(* CoDeSys 2.3.9.41 project: testmodbus.pro *)
(* Libraries: Util.lib 18.5.10 15:14:28, ПЛК_ПЧВ_v2.lib 26.7.19 14:18:06, STANDARD.LIB 4.10.05 11:14:46, IECSFC.LIB 13.4.06 15:51:28, ANALYZATION.LIB 5.10.99 09:05:06 *)

(* PLC configuration (modules and I/O channels)
InputByte AT %IB0.0 [ByteInput] 8 discrete inputs
Discrete output 2 bit [ID101] node 1, in %IB1 out %QB1 {PinCount = 2; SafeValueBool = FALSE; SafeValueBool = FALSE; Visibility = No}
  DO_1_0 AT %QX1.0 [BitOutput] First
  DO_1_1 AT %QX1.1 [BitOutput] Second
Discrete output 2 bit [ID101] node 2, in %IB2 out %QB2 {PinCount = 2; SafeValueBool = FALSE; SafeValueBool = FALSE; Visibility = No}
  DO_2_0 AT %QX2.0 [BitOutput] First
  AT %QX2.1 [BitOutput] Second
Discrete output 2 bit [ID101] node 3, in %IB3 out %QB3 {PinCount = 2; SafeValueBool = FALSE; SafeValueBool = FALSE; Visibility = No}
  DO_3_0 AT %QX3.0 [BitOutput] First
  AT %QX3.1 [BitOutput] Second
Discrete output 2 bit [ID101] node 4, in %IB4 out %QB4 {PinCount = 2; SafeValueBool = FALSE; SafeValueBool = FALSE; Visibility = No}
  DO_4_0 AT %QX4.0 [BitOutput] First
  AT %QX4.1 [BitOutput] Second
Discrete output 2 bit [ID101] node 5, in %IB5 out %QB5 {PinCount = 2; SafeValueBool = FALSE; SafeValueBool = FALSE; Visibility = No}
  DO_5_0 AT %QX5.0 [BitOutput] First
  AT %QX5.1 [BitOutput] Second
Discrete output 2 bit [ID101] node 6, in %IB6 out %QB6 {PinCount = 2; SafeValueBool = FALSE; SafeValueBool = FALSE; Visibility = No}
  DO_6_0 AT %QX6.0 [BitOutput] First
  AT %QX6.1 [BitOutput] Second
Special output [ID104] node 7, in %IB7 out %QB7 {Visibility = No; PinCount = 1}
  AT %QX7.0 [BitOutput] Special output
ModBus (Master) [MODBUS_MASTER_ID450] node 8, in %IB8 out %QB8 {Visibility = No}
  modbusLastAddr AT %QD8.0 [DWordOutput] Last address
  modbusLastErr AT %QW8.1 [WordOutput] Last error
  RS-485-1 [COM1_USART] node 0, in %IB8.0 out %QB8.0 {CommunicationSpeed = 19200; Parity = NO PARITY CHECK; BitLength = 8 bits; StopLength = One stop bit; InterfaceType = RS485; FrameOriented = RTU; Timeout = 0; Visibility = No}
  Universal Modbus device [ID2000] node 1, in %IB8.1 out %QB8.1 {ModuleIP = 10:0:0:223; ServiceTimeout = 150; TCPport = 502; NetMode = Serial; ModuleSlaveAddress = 2; RequestType = By poll time; PeriodOfService = 1000; Visibility = No; RepeatCounter = 2; ByteSequence = Native}
    AT %QB8.1.0 [ComChannel] Command (0xff - Start)
Dist_on_pistol_1 AT %IW8.1.0.0 [WordInput]
Dist_on_pistol_2 AT %IW8.1.1.0 [WordInput]
Dist_on_pistol_3 AT %IW8.1.2.0 [WordInput]
Dist_on_pistol_4 AT %IW8.1.3.0 [WordInput]
Dist_on_pistol_5 AT %IW8.1.4.0 [WordInput]
Dist_on_pistol_6 AT %IW8.1.5.0 [WordInput]
Dist_on_pistol_7 AT %IW8.1.6.0 [WordInput]
Dist_on_pistol_8 AT %IW8.1.7.0 [WordInput]
Dist_off_pistol_1 AT %IW8.1.8.0 [WordInput]
Dist_off_pistol_2 AT %IW8.1.9.0 [WordInput]
Dist_off_pistol_3 AT %IW8.1.10.0 [WordInput]
Dist_off_pistol_4 AT %IW8.1.11.0 [WordInput]
Dist_off_pistol_5 AT %IW8.1.12.0 [WordInput]
Dist_off_pistol_6 AT %IW8.1.13.0 [WordInput]
Dist_off_pistol_7 AT %IW8.1.14.0 [WordInput]
Dist_off_pistol_8 AT %IW8.1.15.0 [WordInput]
DistOnPistMinimum AT %IW8.1.16.0 [WordInput]
qInvStatusW AT %QW8.1.17.0 [WordOutput]
Universal Modbus device [ID2000] node 2, in %IB8.2 out %QB8.2 {ModuleIP = 10:0:0:223; ServiceTimeout = 150; TCPport = 502; NetMode = Serial; ModuleSlaveAddress = 2; RequestType = By poll time; PeriodOfService = 1500; Visibility = No; RepeatCounter = 2; ByteSequence = Native}
  AT %QB8.2.0 [ComChannel] Command (0xff - Start)
iTP1 AT %IW8.2.0.0 [WordInput]
iTP2 AT %IW8.2.1.0 [WordInput]
iTP3 AT %IW8.2.2.0 [WordInput]
iTP4 AT %IW8.2.3.0 [WordInput]
iTP5 AT %IW8.2.4.0 [WordInput]
iTP6 AT %IW8.2.5.0 [WordInput]
iTP7 AT %IW8.2.6.0 [WordInput]
iTP8 AT %IW8.2.7.0 [WordInput]
iTPGlob AT %ID8.2.8.0 [FloatInput]
Universal Modbus device [ID2000] node 3, in %IB8.3 out %QB8.3 {ModuleIP = 10:0:0:223; ServiceTimeout = 150; TCPport = 502; NetMode = Serial; ModuleSlaveAddress = 2; RequestType = By poll time; PeriodOfService = 700; Visibility = No; RepeatCounter = 2; ByteSequence = Native}
  AT %QB8.3.0 [ComChannel] Command (0xff - Start)
task_speed_panel_real AT %ID8.3.0.0 [FloatInput]
speed_at_50Hz AT %ID8.3.1.0 [FloatInput]
speed_at_25Hz AT %ID8.3.2.0 [FloatInput]
speed_Max_panel AT %ID8.3.3.0 [FloatInput]
speed_Min_panel AT %ID8.3.4.0 [FloatInput]
qDetR AT %ID8.3.5.0 [FloatInput]
qMetR AT %ID8.3.6.0 [FloatInput]
follow_Sign_Loss AT %IW8.3.7.0 [WordInput]
qMaxDetLen AT %IW8.3.8.0 [WordInput]
qVersion AT %QD8.3.9.0 [FloatOutput]
Universal Modbus device [ID2000] node 4, in %IB8.4 out %QB8.4 {ModuleIP = 10:0:0:223; ServiceTimeout = 150; TCPport = 502; NetMode = Serial; ModuleSlaveAddress = 2; RequestType = By value change; PeriodOfService = 100; Visibility = No; RepeatCounter = 2; ByteSequence = Native}
  AT %QB8.4.0 [ComChannel] Command (0xff - Start)
qInputB_DO1_6 AT %QW8.4.0.0 [WordOutput]
Universal Modbus device [ID2000] node 5, in %IB8.5 out %QB8.5 {ModuleIP = 10:0:0:223; ServiceTimeout = 150; TCPport = 502; NetMode = Serial; ModuleSlaveAddress = 2; RequestType = By poll time; PeriodOfService = 200; Visibility = No; RepeatCounter = 2; ByteSequence = Native}
  AT %QB8.5.0 [ComChannel] Command (0xff - Start)
qStatusW AT %QW8.5.0.0 [WordOutput]
controlPing AT %ID8.5.1.0 [FloatInput]
qDet_met AT %QD8.5.2.0 [FloatOutput]
qDet_Cnt AT %QD8.5.3.0 [FloatOutput]
controlPong AT %QD8.5.4.0 [FloatOutput]
qAbuseW AT %IW8.5.5.0 [WordInput]
qlast_Det_Len AT %QD8.5.6.0 [FloatOutput]
qlast_Det_Time AT %QD8.5.7.0 [FloatOutput]
AT %QB8.6.0 [ComChannel] Command (0xff - Start)
Status_word AT %IW8.6.0.0 [WordInput]
Frequency AT %IW8.6.1.0 [WordInput]
Power AT %IW8.6.2.0 [WordInput]
Voltage AT %IW8.6.3.0 [WordInput]
Current AT %IW8.6.4.0 [WordInput]
Inv_Error AT %ID8.6.5.0 [DWordInput]
Minimum_frequency AT %IW8.6.6.0 [WordInput]
Maximum_frequency AT %IW8.6.7.0 [WordInput]
Command_word AT %QW8.6.8.0 [WordOutput]
Task_RS485 AT %IW8.6.9.0 [WordInput]
Set_Speed AT %QW8.6.10.0 [WordOutput] 0-16384
Set_MinTask AT %QD8.6.11.0 [DWordOutput]
Set_MaxTask AT %QD8.6.12.0 [DWordOutput]
*)

(* Task configuration *)
TASK cycle_counters (PRIORITY := 0, INTERVAL := T#5ms);
	counters();
END_TASK
TASK main_task (PRIORITY := 1); (* freewheeling *)
	PLC_PRG();
END_TASK

(* Global variable list: Global_Variables *)
VAR_GLOBAL
	total_cycles: DWORD;
	details_meters: REAL;			(*прошло деталей в метрах - берётся от длины в мм*)
	contr_StatusW:  WORD;   			(*статусное слово контроллера - заполняем в главном цикле*)
	contr_AbuseW: WORD;			(*командное слово контроллера - отрабатывает в главном цикле*)
       needSynhro : BOOL := TRUE;	(*Если требуется синхронизация - конвейер не обрабатывает команды управления*)
	freeCounters: BOOL := TRUE;	(*приказ очистить массив счетчика и ВЫКЛючить Пистолеты*)
	last_Limit_switch_part: BOOL := FALSE; (*предыдущее значение датчика детали*)
	last_Det_length: REAL := 0.0;
	last_Det_Time: REAL := 0.0;		(*последнее время на деталь в миллисекундах*)
	version: REAL := 0.6;
	pist: ARRAY[1..4] OF BOOL;
END_VAR

VAR_GLOBAL   (*переменные ошибок*)
	errSensor: BOOL := FALSE; 		(* вырабатывается если количество деталей превысило Максимум или слишком длинная деталь *)
										(* пока активна ошибка - не будут накапливаться данные о деталях, пистолеты выключатся*)
	errTaskSpeed: BOOL := FALSE; 	(* вырабатывается если значение скорости не в диапазоне макс/мин или равно 0 *)

END_VAR

VAR_GLOBAL
	(*Входы контроллера*)
	Start_conveyor: BOOL;    			(*DI_1 Включить конвейер *)
	Stop_conveyor: BOOL;   			(*DI_2 Выключить конвейер *)
	Following_machine: BOOL;   		(*DI_3 Сигнал от следующей машины*)
	Fan_on: BOOL;					(*DI_4 Вытяжка включена*)
	(*Pistols_automat_mode: BOOL;	Пистолеты в автоматическом режиме*)
	Door_Closed: BOOL;				(*DI_5 Концевой выключатель двери*)
	Limit_switch_part: BOOL;			(*DI_6 Концевой выключатель наличия детали*)
	Pistols_5_8_run: BOOL;			(*DI_7 Включены пистолеты 5-8*)

	(*Выходы контроллера*)
	Conveyor_green: BOOL;                     (*Конвейер готов к включению (сигнальная лампа) *)
	Conveyor_runNow: BOOL;			(*Конвейер поехал,сигнал на предыдущую машину *)

END_VAR

VAR_GLOBAL RETAIN PERSISTENT (*эти данные хранятся в энергонезависимой памяти*)
	details_count: REAL;				(*Счётчик кол-ва деталей. Сбрасывается по команде с панели *)
	details_mMeters: REAL;			(*Счётчик общей длины детали в мм, сбрасывается с панели *)
	details_Real_mMeters: REAL;	(*Необнуляемый счётчик  общей длины детали в мм*)
END_VAR

(* POU counters, ST *)
PROGRAM counters
VAR CONSTANT
	MAXDETCNT:INT:= 10;
END_VAR

VAR
	cycleinterval_ms: REAL := 4.99; (*такой установлен в конфигураторе задач !!!!!!!!!!!!!!!!!!!!!!!!!!!!!!!!!!!!!!!!!!!!!!!!!!!!!!!!!!!!!!!!!!!!*)

   (*    cycleinterval_ms_calc: REAL;
	lasttime: TIME;
	total_cycles_loss: DWORD; *)

	cycle_mm: REAL; (*надо пересчитать в мм на текущий момент времени в зависимости от скорости погонажки*)
	Counter: ARRAY[1..4, 0..1, 0..MAXDETCNT] OF REAL; (* 4 pistools, On(0), Off(1), push counter     in mm ! *)
	PistLen: ARRAY[1..4,0..1] OF INT; (*4 pist, 0 - Up Len, 1 - UpLen+Off Len *)
	PistTime: ARRAY[1..4] OF INT; (*время предварительного срабатывания пистолета - пересчёт в мм*)
	i,j,k: INT;
	detOn: BOOL;
	detOff: BOOL;
	need_Pistols_On: BOOL;
END_VAR
(*программа выполняется с частотой вызовов 1 раз в 5 мсек*)
(*m/min > *)
(*cycleinterval_ms_calc := TIME_TO_REAL(TIME()-lastTime)+0.01;
lastTime := TIME();*)
(*
CycleTime_100mks;
CPU_OverLoaded;

total_cycles := total_cycles+1;
total_cycles_loss := total_cycles_loss + BOOL_TO_DWORD( cycleinterval_ms <> cycleInterval_ms_calc);
*)
cycle_mm := task_speed_panel_real*1000/60/(1000/cycleinterval_ms);

	FOR i := 1 TO 4 DO
	FOR j := 0 TO 1 DO
		FOR k:=0 TO MAXDETCNT DO
			IF freecounters THEN
				Counter[i,j,k] := 0.0;
			END_IF;
		END_FOR
	END_FOR
	IF freecounters THEN
		Counter[i,1,0] := 0.001; (*выключить пистолет*)
	END_IF;
	END_FOR
	freecounters := FALSE;

Limit_switch_part:=DI_6 AND NOT errSensor; 	(*Концевой выключатель наличия детали причём если нет его ошибки*)
Pistols_5_8_run:=DI_7; 	(*Включены пистолеты 5-8*)

(*прошел цикл, значит пора сократить все длины на cycle_mm, заодно разобраться с включением выключением,
а потом уже сделать перенос величин ставших менее 0.0*)

FOR i := 1 TO 4 DO
	FOR j := 0 TO 1 DO
		FOR k:=0 TO MAXDETCNT DO
			IF Counter[i,j,k] <> 0.0 THEN
				Counter[i,j,k] := Counter[i,j,k]-cycle_mm;
			END_IF;
		END_FOR
	END_FOR
								  (* СПЕРВА ВЫКЛЮЧИМ, ПОТОМ ВКЛЮЧИМ - убираем пересечения *)
	IF (Counter[i,1,0] < 0)  THEN (*начало  цикла (голова) в нуле. если нулевое стало меньше 1 - выключим пистолет, но не если есть след.деталь*)
		pist[i] := FALSE;
	END_IF;
	IF Counter[i,0,0] < 0 THEN (*начало  цикла (голова) в нуле. если нулевое стало меньше 0 - включим пистолет*)
		pist[i] := TRUE;
	END_IF;
END_FOR

detOn := FALSE;
detOff := FALSE;

IF NOT last_Limit_switch_part AND Limit_switch_part THEN (*деталь началась*)
	detOn := TRUE;
	last_Det_length := 0.0;
	last_Det_time := 0.0;
END_IF;

IF last_Limit_switch_part AND NOT Limit_switch_part THEN (*деталь прошла*)
	details_count := details_count +1;
	qLast_Det_time := last_Det_time;
	detOff := TRUE;
END_IF;

IF Limit_switch_part THEN (*если концевик показывает деталь - увеличим погонаж*)
	details_mMeters := details_mMeters+cycle_mm;
	details_Real_mMeters := details_Real_mMeters +cycle_mm;
	last_Det_Length := last_Det_Length+cycle_mm;
	last_Det_Time := last_Det_Time + cycleinterval_ms;
	IF last_Det_Length > qmaxDetLen THEN
		errSensor := TRUE;
	END_IF;
END_IF;
details_meters := details_mMeters / 1000;

(* заполнить массив включения выключения если не синхронизация *)
IF NOT needSynhro THEN
IF NOT Pistols_5_8_run THEN
   PistLen[1,0] := Dist_on_pistol_1; PistLen[1,1] := Dist_off_pistol_1;
   PistLen[2,0] := Dist_on_pistol_2; PistLen[2,1] := Dist_off_pistol_2;
   PistLen[3,0] := Dist_on_pistol_3; PistLen[3,1] := Dist_off_pistol_3;
   PistLen[4,0] := Dist_on_pistol_4; PistLen[4,1] := Dist_off_pistol_4;
	PistTime[1] := REAL_TO_INT((-INT_TO_REAL(iTP1)+iTPGlob)*cycle_mm/cycleinterval_ms);
	PistTime[2] := REAL_TO_INT((-INT_TO_REAL(iTP2)+iTPGlob)*cycle_mm/cycleinterval_ms);
	PistTime[3] := REAL_TO_INT((-INT_TO_REAL(iTP3)+iTPGlob)*cycle_mm/cycleinterval_ms);
	PistTime[4] := REAL_TO_INT((-INT_TO_REAL(iTP4)+iTPGlob)*cycle_mm/cycleinterval_ms);
ELSE
   PistLen[1,0] := Dist_on_pistol_5; PistLen[1,1] := Dist_off_pistol_5;
   PistLen[2,0] := Dist_on_pistol_6; PistLen[2,1] := Dist_off_pistol_6;
   PistLen[3,0] := Dist_on_pistol_7; PistLen[3,1] := Dist_off_pistol_7;
   PistLen[4,0] := Dist_on_pistol_8; PistLen[4,1] := Dist_off_pistol_8;
	PistTime[1] := REAL_TO_INT((-INT_TO_REAL(iTP5)+iTPGlob)*cycle_mm/cycleinterval_ms);
	PistTime[2] := REAL_TO_INT((-INT_TO_REAL(iTP6)+iTPGlob)*cycle_mm/cycleinterval_ms);
	PistTime[3] := REAL_TO_INT((-INT_TO_REAL(iTP7)+iTPGlob)*cycle_mm/cycleinterval_ms);
	PistTime[4] := REAL_TO_INT((-INT_TO_REAL(iTP8)+iTPGlob)*cycle_mm/cycleinterval_ms);
END_IF;

FOR i := 1 TO 4 DO
IF PistLen[i,0] > 0 THEN (*хоть какая-то длина указана, ок*)
   PistLen [i,0] := PistLen[i,0] + PistTime[i];
   IF PistLen[i,0] <=0 THEN PistLen[i,0] := 1;END_IF;
   PistLen[i,1] := PistLen[i,0] + PistLen[i,1];
END_IF;
END_FOR;

END_IF;

(*прокрутить списки деталей*)

FOR i := 1 TO 4 DO
	j := 0;
	IF Counter[i,j,0] < INT_TO_REAL( PistLen[i,0] - PistLen[i,1])-5.0 THEN (*убрать деталь*)
		FOR k:=0 TO MAXDETCNT-1 DO (*-1, т.к. [,,k] элемент = 0, удобненько*)
			Counter[i,j,k] := Counter[i,j,k+1];
		END_FOR
	END_IF
END_FOR

FOR i := 1 TO 4 DO
	j := 1;
	IF Counter[i,j,0] < 0 THEN (*убрать деталь*)
		FOR k:=0 TO MAXDETCNT-1 DO (*-1, т.к. [,,k] элемент = 0, удобненько*)
			Counter[i,j,k] := Counter[i,j,k+1];
		END_FOR
	END_IF
END_FOR

(*добавить деталь если началась*)
IF detOn THEN
	FOR i := 1 TO 4 DO
	 j := 0;
	FOR k:=0 TO MAXDETCNT-1 DO
		IF Counter[i,j,k] = 0.0 THEN
			EXIT;
		END_IF;
	END_FOR
	(*хочется не добавлять если k - крайний и выработать ошибку*)
	IF k=MAXDETCNT THEN
		errSensor := TRUE;
	ELSE
		Counter[i,j,k] := PistLen[i,0]; (*значение ожидания до включения если оно больше чем DistOnPistMinimum*)
		IF PistLen[i,0] < DistOnPistMinimum THEN  Counter[i,j,k] := 0.0; END_IF;
	END_IF;
	END_FOR
END_IF;

(*добавить конец детали деталь если кончилась*)
IF detOff THEN
	FOR i := 1 TO 4 DO
	 j := 1;
	FOR k:=0 TO MAXDETCNT-1 DO
		IF Counter[i,j,k] = 0.0 THEN
			EXIT;
		END_IF;
	END_FOR
	(*хочется не добавлять если k - крайний и выработать ошибку*)
	IF k=MAXDETCNT THEN
		errSensor := TRUE;
	ELSE
		IF (k > 0) AND (PistLen[i,0] < REAL_TO_INT(Counter[i,j,k-1]) ) THEN (*более 1 детали и перекрывает расстояние, правим предыдущую*)
		   k := k-1;
		END_IF;
		Counter[i,j,k] := PistLen[i,1]; (*значение ожидания до выключения если включение больше чем DistOnPistMinimum*)
		IF PistLen[i,0] < DistOnPistMinimum THEN  Counter[i,j,k] := 0.0; END_IF;
	END_IF;
	END_FOR
END_IF;

need_Pistols_On := contr_abuseW.1  AND Door_Closed AND Fan_on; (*просит включить распыление и ВЫтяжка *)

(*включить/выключить пистолеты *)
DO_3_0 := pist[1] OR need_Pistols_On;
DO_4_0 := pist[2] OR need_Pistols_On;
DO_5_0 := pist[3] OR need_Pistols_On;
DO_6_0 := pist[4] OR need_Pistols_On;

(*запомнить состояние детали*)
last_Limit_switch_part := Limit_switch_part;
END_PROGRAM

(* POU PLC_PRG, ST *)
PROGRAM PLC_PRG
VAR
	synhroW: DWORD := 0;

	com_word: com_word_fb;
	Invertor_stop: BOOL := FALSE;
	Invertor_start: BOOL := FALSE;
	Invertor_reverse:BOOL := FALSE;
	Invertor_speed_ok: BOOL := FALSE;

(*переменные объединяющиес текущий статус контроллера*)
	Invertor_Pwr_On: BOOL := FALSE; (*инвертор найден по шине, получен статус отличный от 0 и он в автомате и готов*)
	Conveyor_On: BOOL; (*включен двигатель конвейера*)

(*просто какие-то временные переменные*)
	w1: WORD;
	dw, mit, mat: DWORD;
	bol: BOOL;
	b: REAL;
	k: REAL;
	modbusInvLastErr: WORD := 0;

(* Статус частотника *)
	stat_word: stat_word_fb;

	Invertor_alarm: BOOL;		(* Авария частотника *)
	Invertor_warning: BOOL; 		(* Предупреждение частотника *)
	Invertor_auto: BOOL;			(* Частотник в автоматическом режиме *)
	Invertor_work: BOOL; 			(* Частотник в работе *)

(*переменные для управления ПЧВ*)
	rsp : REAL;
	abuse_50Hz: BOOL; (*принуждает ПЧВ запустить двигатель на 50 Hz*)
	abuse_25Hz: BOOL; (*принуждает ПЧВ запустить двигатель на 25 Hz*)
	frequency_Equal: BOOL := FALSE;
	lastFreqReqw: WORD := 0;
	task_invertor: task_fb;

(*FB logic*)

	Run:BOOL;
	Stop:BOOL;
	Common_Alarm: BOOL;
	R_TRIG: R_TRIG;
	F_TRIG: F_TRIG;
	F_TRIG1: F_TRIG;
	RS1: RS;

END_VAR
(*проверка связи по модбасу с ПЧВ Addr=1 *)
IF  modbusLastAddr = 1 THEN
	modbusInvLastErr := modbusLastErr;
END_IF;

(*Статус частотника*)
stat_word(
	stat_word:= Status_word,
	ready_engine=> ,
	ready_drvive=> ,
	slow_stop_stat=> ,
	alarm=>Invertor_alarm ,
	warning=> Invertor_warning,
	task_stat=>Invertor_speed_ok ,
	avt=>Invertor_auto ,
	over_range=> ,
	work_stat=>Invertor_work ,
	voltage=> ,
	current=> ,
	heat=> );

Invertor_Pwr_On := (Status_Word > 0) AND (modbusInvLastErr = 0) AND Invertor_auto AND NOT Invertor_alarm;


Start_conveyor:=DI_1 ;	(*Включение конвейера*)
Stop_conveyor:=NOT DI_2 ; 	(*Отключение конвейера*)
Following_machine:=DI_3; (*Сигнал от предыдущей машины*)
Fan_on:=DI_4; 			(*Вытяжка включена*)
Door_closed := NOT DI_5; 		(*Дверь закрыта наоборот )) *)
Pistols_5_8_run := DI_7; (*выбраны 5-8 пистолеты*)

errTaskSpeed :=  	(task_speed_panel_real <= 0) OR
					(speed_at_50Hz <= 0) OR
					(speed_at_50Hz <= speed_at_25Hz) OR
					(speed_Max_panel <= speed_Min_panel) OR
					(speed_Max_panel <= 0) OR
					(task_speed_panel_real > speed_Max_panel) OR
					(task_speed_panel_real < speed_Min_panel);

Conveyor_On := Invertor_Work;

(*посчитаем - выставил ли частотник реальную частоту*)
w1 := (100*(100*Frequency+1)) / (100*lastFreqReqw+1);
frequency_Equal := Invertor_Work AND ((w1 > 97) OR Invertor_speed_ok);    (*скорость соответствует на 98% и более*)

(*программируем общую логику*)
(*надо получить состояние, зажечь лампу, дать сигнал на машину*)

(*работа зависит от    			 follow_Sign_Loss *)

R_TRIG
(CLK:=Start_conveyor, 		(*Выделение переднего фронта на запуск конвейера*)
 Q=>Run );

F_TRIG
(CLK:=Stop_conveyor,			(*Выделение переднего фронта на останов конвейера*)
 Q=>Stop );

Common_Alarm := errSensor OR errTaskSpeed OR Invertor_Alarm OR NOT Invertor_Pwr_On ;

RS1(
SET:= ( Fan_On AND Run  AND Invertor_Pwr_On AND Door_Closed),
RESET1:= (Stop OR NOT Fan_On OR NOT Door_Closed OR Common_alarm),
Q1=> Conveyor_green);

IF Conveyor_green THEN (*есть базовое разрешение на включение, проверим логику с ведомой машиной*)
   Conveyor_runNow := Following_machine; (*запустить конвейер по сигналу от след машины*)
IF follow_Sign_Loss > 0 THEN (*определено ждать*)
  ;
   (*помигаем лампочкой если нет машины*)
   (*мигать будем потом там внизу*)
ELSE (*определено закончить работу*)
   Conveyor_green := Following_machine;
END_IF;
ELSE (*конвейер не зелёный*)
   Conveyor_runNow := FALSE;
END_IF;

Invertor_start:=Conveyor_runNow;

(*задний фронт на останов частотника используем для обнуления массива*)
F_TRIG1(
	CLK:=Conveyor_runNow ,
	Q=> Invertor_stop);

IF Conveyor_green AND NOT Following_machine THEN (*замигаем лампу*)
   DO_1_0 := TIME_TO_DWORD(TIME()) MOD 1000 > 500;
ELSE
    DO_1_0:=Conveyor_green;  (*сигнальная лампа*)
END_IF;
DO_2_0:=Conveyor_runNow;  (*Конвейер включен(,сигнал на предыдущую машину)*)

(* создание слова статуса контроллера*)

contr_statusW.0  := 1; (*контроллер под питанием*)
contr_statusW.1 := Invertor_Pwr_On;
contr_statusW.2 := Fan_On;
contr_statusW.3 := Conveyor_On;
contr_statusW.4 := Door_Closed;
contr_statusW.5 := Following_machine;
contr_statusW.6 := Pistols_5_8_run;
contr_statusW.7 := Conveyor_runNow;
contr_statusW.8 := errSensor;
contr_statusW.9 := errTaskSpeed;
contr_statusW.10 := Invertor_Alarm;

(*Загрузить возможные переменные с подчиненных устройств
 и проверить контрольную сумму. предварительно её рассчитав.

выставит needSynhro - что означает не все данные загружены
требуется синхронизация!
*)

freeCounters := errSensor OR NOT Door_Closed OR NOT fan_on OR Invertor_stop; (* если ошибка сенсора или дверь не закрыта -  очистить список деталей *)

synhroW :=
	Dist_on_pistol_1+Dist_off_pistol_1+
	Dist_on_pistol_2+Dist_off_pistol_2+
	Dist_on_pistol_3+Dist_off_pistol_3+
	Dist_on_pistol_4+Dist_off_pistol_4+
	Dist_on_pistol_5+Dist_off_pistol_5+
	Dist_on_pistol_6+Dist_off_pistol_6+
	Dist_on_pistol_7+Dist_off_pistol_7+
	Dist_on_pistol_8+Dist_off_pistol_8+
	follow_Sign_Loss+
	TRUNC(10*task_speed_panel_real)+
	TRUNC(10*speed_at_50Hz)+
	TRUNC(10*speed_Max_panel)+
	TRUNC(10*speed_Min_panel)+
	qMaxDetLen+
	DistOnPistMinimum+
	TRUNC(10*speed_at_25Hz)+
	iTP1+iTP2+iTP3+iTP4+iTP5+iTP6+iTP7+iTP8+
	TRUNC(10*ABS(iTPGlob));


controlPong := DWORD_TO_REAL(synhroW);
needSynhro :=  controlPing <> controlPong; (* установить необходимость синхронизации*)

contr_abuseW := qAbuseW;
needSynhro := needSynhro OR contr_abuseW.0; (*проверить не прислала ли панелька своё требование синхронизации*)

IF contr_abuseW.2 THEN (*bit 2 просит обнулить счётчики*)
	Details_Count := 0;
	Details_mMeters := 0;
END_IF;
IF contr_abuseW.3 THEN (*bit 3 просит установить счётчики*)
	Details_Count := qDetR;
	Details_mMeters := qMetR*1000;
END_IF;
IF contr_abuseW.4 THEN (*bit 4 просит сбросить ошибки*)
	errSensor := FALSE;       (* сбросим ошибку сенсора, мало ли .... исправит ситуацию*)
END_IF;
abuse_50Hz := contr_abuseW.5; (*bit 5 установить скорость 50 Hz*)
abuse_25Hz := contr_abuseW.6; (*bit 6 установить скорость 25 Hz*)

(* заполнить основные переменные для передачи в панельки.
передача 3 раза в сек *)

qStatusW := contr_StatusW;
qDet_Cnt := Details_Count;
qDet_Met := Details_Meters;
qLast_det_len := last_Det_Length;
qInvStatusW := status_word;

w1 := SHL(InputByte,8); w1.0 := DO_1_0; w1.1 := DO_2_0; w1.2 := DO_3_0; w1.3 := DO_4_0; w1.4 := DO_5_0; w1.5 := DO_6_0;
w1.6 := frequency_Equal;
qInputB_DO1_6 := w1;
qVersion := Version;

(*программируем ПЧВ*)
(*проверяем на ошибки и если всё ок - начинаем им управлять*)
	w1 := Task_RS485; (*0-16384*)

	IF NOT errTaskSpeed AND NOT needSynhro THEN (*вычисляем какую скорость поставить*)
		(*запрограммируем линейность по 2 точкам   ??? *)
		k := (50-25) / (speed_at_50Hz - speed_at_25Hz);
		b := 50-k*speed_at_50Hz;
		rsp := task_speed_panel_real * k + b; (*???*) (*rsp = необходимая частота Hz*)
		(*предыдущая версия расчёта по 1 коэффициенту*)
(*		rsp := task_speed_panel_real / speed_at_50Hz * 50; (*rsp = необходимая частота Hz*) *)

		w1 := REAL_TO_WORD(rsp*10); (*w1 теперь соответсвует частоте * 10 как и в мин, макс*)
		IF w1 < Minimum_frequency THEN w1 := Minimum_frequency; END_IF;
		IF w1 > Maximum_frequency THEN w1 := Maximum_frequency; END_IF;
		(*Maximum_frequency (*650   = 65Гц*)*)
		lastFreqReqw := w1;
		(*на этом этапе w1 : [0..650] НАДО конвертнуть в 0 - 16384*)
		rsp := 16384 * w1 / Maximum_frequency;
		w1 := REAL_TO_WORD(rsp);
	END_IF;
	IF errTaskSpeed AND NOT needSynhro THEN
		invertor_Start := FALSE;
	END_IF;

	bol := FALSE;
	IF NOT needSynhro AND (abuse_50Hz OR abuse_25Hz) THEN (*принудим двигатель раскрутиться на 50 hz*)
		w1 := 500;
		IF abuse_25Hz THEN w1 := 250; END_IF;
		lastFreqReqw := w1;
		(*на этом этапе w1 = 500|250  НАДО конвертнуть в 0 - 16384*)
		rsp := 16384 * w1 / Maximum_frequency;
		w1 := REAL_TO_WORD(rsp);
		bol := (w1 > 0);
	END_IF;
       Set_MinTask := Minimum_frequency * 100;
	Set_MaxTask := Maximum_frequency * 100;
	Set_Speed := w1; (*0-16384*)


(*task_invertor(
	t_min:=task_frequency_min ,
	t_max:=task_frequency_max ,
	task_value:=task_frequency_invertor ,
	pre_task_value1:= ,
	pre_task_value2:=,
	pre_task_value3:= ,
	pre_task_value4:= ,
	num_task:= ,
	lim_h:= ,
	Idc_stop_val:= ,
	rs_off:= ,
	task_min=>mit ,
	task_max=>mat,
	task=>w1 ,
	pre_task_value=> ,
	pre_task_num=> ,
	lim_high=> ,
	Idc_stop=> ,
	rs_out=> );
*)
(*запустить двигатель*)
com_word(
	pre_task_num:= ,
	dc_stop:= ,
	slow_stop:=Invertor_stop ,
	fast_stop:= ,
	start:= Invertor_start OR bol,
	REVERSE:=Invertor_reverse ,
	com_word=>Command_word );
END_PROGRAM

(* POU send_by_modbus, ST *)
PROGRAM send_by_modbus
VAR
   LastAddress AT %QD8.0: DWORD;
   LastError AT %QW8.1: WORD;
   StartPanel AT %QB8.1.0: BYTE;
   StartPanel2 AT %QB8.2.0: BYTE;
   StartInvertor  AT %QB8.3.0: BYTE;
   NextDev : BYTE := 0;
	s1: BYTE;
	s2 :BYTE;
	s3:BYTE;
END_VAR
(* запускается раз в 100 мс *)

s1 := StartPanel; s2 := StartPanel2; s3 := StartInvertor;

(*

s1 := StartPanel; s2 := StartPanel2; s3 := StartInvertor;
IF (NeedSynhro) AND (NextDev = 0) AND  (s1=s2) AND (S1=S3) THEN (*опрос всех данных панельки*)
	StartPanel := 255;
	NextDev := NextDev + 1;
END_IF;

s1 := StartPanel; s2 := StartPanel2; s3 := StartInvertor;
IF (NextDev = 1) AND  (s1=s2) AND (S1=S3) THEN (*миниопрос панельки*)
	StartPanel2 := 255;
	NextDev := NextDev + 1;
END_IF;

s1 := StartPanel; s2 := StartPanel2; s3 := StartInvertor;
IF (NextDev = 2) AND  (s1=s2) AND (S1=S3) THEN (*опрос частотника*)
    StartInvertor := 255;
    NextDev := NextDev + 1;
END_IF;

IF  (lastaddress = 1) THEN
	mb_inv_ok := (lasterror = 0);
END_IF;
IF  (lastaddress = 2) THEN
	mb_Pan_ok := (lasterror = 0);
END_IF;

nextdev := nextdev+1;

IF nextdev > 2 THEN
	nextdev := nextdev MOD 3;
	StartInvertor := 0;
	StartPanel := 0;
	StartPanel2 := 0;
END_IF;
*)
END_PROGRAM
